FUNCTION_BLOCK DRAWARUCOMARKERS (* Draw Aruco Markers *)
  (* Version 1.0, AN, SWDC RTSoft *)
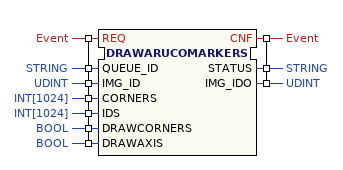
  EVENT_INPUT
    REQ WITH QUEUE_ID, IMG_ID, CORNERS, IDS, DRAWCORNERS, DRAWAXIS;
  END_EVENT
  EVENT_OUTPUT
    CNF WITH STATUS, IMG_IDO;
  END_EVENT
  VAR_INPUT
    QUEUE_ID : STRING;
    IMG_ID : UDINT;
    CORNERS : ARRAY [0..1023] OF INT; (* Array of corner points *)
    IDS : ARRAY [0..1023] OF INT; (* Array of marker IDs *)
    DRAWCORNERS : BOOL; (* Bool flag to Draw Corners *)
    DRAWAXIS : BOOL; (* Bool flag to Draw Axis *)
  END_VAR
  VAR_OUTPUT
    STATUS : STRING;
    IMG_IDO : UDINT;
  END_VAR
  ALGORITHM REQ IN ST:

  END_ALGORITHM
END_FUNCTION_BLOCK
